{attribute 'GeneratedUsingTerminal: KL9191'}
{attribute addProperty BoxType "KL9191"}
{attribute addProperty Id "Contact_DI1AT %I*BOOL0Contact_DI2AT %I*BOOL0Contact_DI3AT %I*BOOL0LED_DO1AT %Q*BOOL0Relay_2kWAT %Q*BOOL0Relay_FAN1AT %Q*BOOL0Relay_FAN2AT %Q*BOOL0Relay_FAN3AT %Q*BOOL0TRIAC_Y1AT %Q*BOOL0TRIAC_Y2AT %Q*BOOL0"}
{attribute addProperty CRC "1193257564"}
{attribute addProperty Size "0"}
TYPE Channel_471FAA5C :
STRUCT
	{attribute addProperty Name "Contact_DI1"}
	Contact_DI1 AT %I* : BOOL;
	{attribute addProperty Name "Contact_DI2"}
	Contact_DI2 AT %I* : BOOL;
	{attribute addProperty Name "Contact_DI3"}
	Contact_DI3 AT %I* : BOOL;
	{attribute addProperty Name "LED_DO1"}
	LED_DO1 AT %Q* : BOOL;
	{attribute addProperty Name "Relay_2kW"}
	Relay_2kW AT %Q* : BOOL;
	{attribute addProperty Name "Relay_FAN1"}
	Relay_FAN1 AT %Q* : BOOL;
	{attribute addProperty Name "Relay_FAN2"}
	Relay_FAN2 AT %Q* : BOOL;
	{attribute addProperty Name "Relay_FAN3"}
	Relay_FAN3 AT %Q* : BOOL;
	{attribute addProperty Name "TRIAC_Y1"}
	TRIAC_Y1 AT %Q* : BOOL;
	{attribute addProperty Name "TRIAC_Y2"}
	TRIAC_Y2 AT %Q* : BOOL;
END_STRUCT
END_TYPE

(* stored: Version 1.2.0.0, ProductVersion 3.1.4024.9
   DUT Channel_471FAA5C: Id {2441912b-f35d-46e1-86a8-bed49578500d} *)
